FUNCTION_BLOCK Stage20 (* Template for a Basic Function Block Type *)
  (* Standard: 61499-2 *)
  (* Version 1.0, 2021-06-20, HP *)
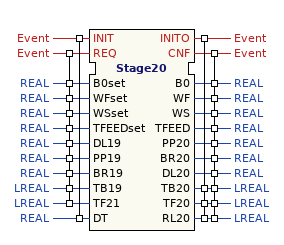
  EVENT_INPUT
    INIT WITH DT; (* Initialization Request *)
    REQ WITH WFset, WSset, TFEEDset, DL19, PP19, BR19, TB19, TF21, B0set; (* Normal Execution Request *)
  END_EVENT
  EVENT_OUTPUT
    INITO WITH TB20, TF20, RL20; (* Initialization Confirm *)
    CNF WITH TB20, DL20, TF20, BR20, PP20, TFEED, WF, WS, RL20, B0; (* Execution Confirmation *)
  END_EVENT
  VAR_INPUT
    B0set : REAL;
    WFset : REAL;
    WSset : REAL;
    TFEEDset : REAL;
    DL19 : REAL;
    PP19 : REAL;
    BR19 : REAL;
    TB19 : LREAL;
    TF21 : LREAL;
    DT : REAL;
  END_VAR
  VAR_OUTPUT
    B0 : REAL;
    WF : REAL;
    WS : REAL;
    TFEED : REAL;
    PP20 : REAL;
    BR20 : REAL;
    DL20 : REAL;
    TB20 : LREAL;
    TF20 : LREAL;
    RL20 : LREAL;
  END_VAR
  VAR
    AB : REAL; (* internal variabel *)
    UU : REAL;
    TREF : REAL;
    AD : REAL;
    AHC : REAL;
    AHR : REAL;
    AS : REAL;
    REC : REAL;
    WN : REAL;
    WN_1 : REAL;
    XKN : REAL;
    C1 : REAL;
    HS : REAL;
    G : REAL;
    W1 : REAL;
    TFREC : REAL;
    TS : REAL;
    DTS : REAL;
    TF20_last : REAL;
    RL20_last : REAL;
    TB20_last : REAL;
    USS : REAL;
    RHOB : REAL;
    CPB : REAL;
    CPF : REAL;
    FMW : REAL;
    HLV : REAL;
    HV : REAL;
    BPR : REAL;
    FMC : REAL;
    U : REAL;
    A : REAL;
    B : REAL;
    C : REAL;
    D1 : REAL;
    d : REAL;
    a : REAL;
    A1 : REAL;
    A2 : REAL;
    A3 : REAL;
    A4 : REAL;
    A5 : REAL;
    A6 : REAL;
    p : REAL;
    q : REAL;
    TC : REAL;
    PC : REAL;
    DTB20 : REAL;
    DEN20 : REAL;
    DH20 : REAL;
    DP20 : REAL;
    DPDH20 : REAL;
    DT20 : REAL;
    m : REAL;
    n : REAL;
    VR20 : REAL;
    DELTA20 : REAL;
    DELTA42 : REAL;
    DELTA64 : REAL;
    DELTA20_last : REAL;
    DELTA42_last : REAL;
    DELTA64_last : REAL;
  END_VAR
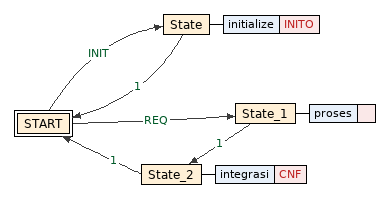
  EC_STATES
    START; (* Initial State *)
    State : initialize -> INITO;
    State_1 : proses;
    State_2 : integrasi -> CNF;
  END_STATES
  EC_TRANSITIONS
    START TO State := INIT;
    State TO START := 1;
    START TO State_1 := REQ;
    State_1 TO State_2 := 1;
    State_2 TO START := 1;
  END_TRANSITIONS
  ALGORITHM initialize IN ST: (* Initialization algorithm *)
TREF :=273.15;
AB :=57.2727;
AHC :=4069.2;
AHR :=2639.7;
AS :=3225.7;
REC :=0.0;
//TF2:=TF2;

//TFEED :=TFEED1+TREF;
 //TS:=TS1+TREF;
WN :=3.0;
XKN :=0.68;
HS:=0.11;
G :=9.81;
W1 :=0.50;

RL20 := 0.632295047243955;
TB20 := 318.010917195497;
TF20 := 314.769851417199;
TF21 := 312.855009206396;


RL20_last :=RL20;
TB20_last :=TB20;
TF20_last :=TF20;
  END_ALGORITHM
  ALGORITHM proses IN ST: (* kalkulasi *)
B0 :=B0set;
WS :=WSset;
TFEED:=TFEEDset;
TFEED:=TFEEDset;
UU := TFEEDset;
U :=UU;

USS :=49.767;
C1 :=0.625;
RHOB :=1032.4; //maassa jenis brine
CPB :=1.00; //heatcapacity Brine
CPF :=1.00; //heat capacity feed
FMW :=23654.0;
HLV :=563.7959;
HV :=625.1971;
BPR :=2.192;
FMC :=34736.09;
//U :=UU; //feed temp



///  Calculate the physical properties

//A :=3.2437814;
//B :=5.86826*0.001;
//C :=1.1702379*0.00000001;
//D1 :=2.1878462*0.001;
//TC :=647.27;
//PC :=218.167;


A1 :=3.2437814;
A2:=5.86826*0.001;
A3:=1.1702379*0.00000001;
A4 :=2.1878462*0.001;
A5 :=647.27;
A6 :=218.167;

DTB20 :=A5-TB20;
DEN20 :=(A1+A2*DTB20+A3*DTB20*DTB20*DTB20)/(1+A4*DTB20)*DTB20/TB20;
p:=DEN20;
q:=10.0;
PP20 :=A6/(EXPT(q, p));

// calculate the brine flow rates
DP20:=PP19-PP20;
DH20:=RL20-C1*HS;
DPDH20 :=DP20*101000+G*RHOB*DH20;
m:=DPDH20*RHOB;
n:=0.5;
BR20 :=WN*XKN*RL20*(EXPT(m, n));
BR20 :=BR20*60.0/1000.0;

// calculate the vapor flow rates

DT20 :=TB20-BPR/1.8-(TF21+TF20)*0.5;
VR20:=U*AHR*DT20/HLV/1000.0;
DL20 :=DL19+VR20;


//// state equation
DELTA20 :=(BR19-BR20-VR20)*1000.0/RHOB/AB;
DELTA42 :=((BR19*CPB*(TB19-TB20))-VR20*(HV-CPB*(TB20-TREF)))*1000.0/AB/RHOB/CPB/RL20;
DELTA64 :=(WF*CPF*(TF21-TF20)*1000+(U*AHR*DT20))/FMW/CPF;
  END_ALGORITHM
  ALGORITHM integrasi IN ST: (* new algorithm *)
B0:=B0set;
WF :=WFset;
WS :=WSset;
TFEED:=TFEEDset;
//integrasi
RL20 := (DELTA20 + DELTA20_last)*0.5*DT + RL20_last;
DELTA20_last :=DELTA20 ;
RL20_last :=RL20;

TB20:= (DELTA42 + DELTA42_last)*0.5*DT + TB20_last;
DELTA42_last :=DELTA42 ;
TB20_last:=TB20;

TF20 := (DELTA64 + DELTA64_last)*0.5*DT + TF20_last;
DELTA64_last :=DELTA64 ;
TF20_last :=TF20;
  END_ALGORITHM
END_FUNCTION_BLOCK
